(* Logix 5000 project; controller SX_V040001_C001 vendor 1 type 14 code 77 rev 16.22; software revision 16.04; part 15 of 35 *)
(* tags used below, declared in another part *)
   G_DInput : DINT[3];
   G_DOutput : DINT[3];
   louvre : INT[11];
   PARAMETER : INT[501];
(* MainProgram, continued *)

ROUTINE Louvre3Position   (* ladder *)
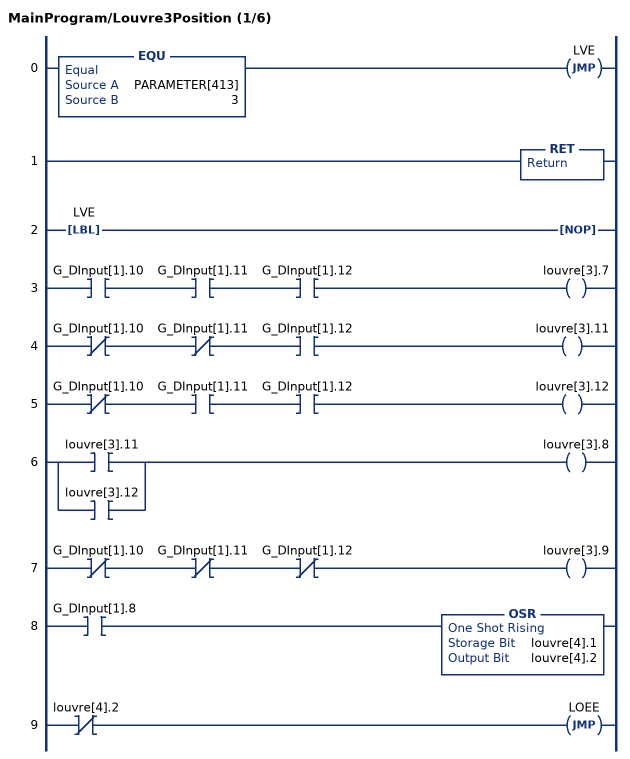
   0: EQU(PARAMETER[413],3)JMP(LVE);
   1: RET();
   2: LBL(LVE)NOP();
   3: XIC(G_DInput[1].10)XIC(G_DInput[1].11)XIC(G_DInput[1].12)OTE(louvre[3].7);
   4: XIO(G_DInput[1].10)XIO(G_DInput[1].11)XIC(G_DInput[1].12)OTE(louvre[3].11);
   5: XIO(G_DInput[1].10)XIC(G_DInput[1].11)XIC(G_DInput[1].12)OTE(louvre[3].12);
   6: [XIC(louvre[3].11) ,XIC(louvre[3].12) ]OTE(louvre[3].8);
   7: XIO(G_DInput[1].10)XIO(G_DInput[1].11)XIO(G_DInput[1].12)OTE(louvre[3].9);
   8: XIC(G_DInput[1].8)OSR(louvre[4].1,louvre[4].2);
   9: XIO(louvre[4].2)JMP(LOEE);
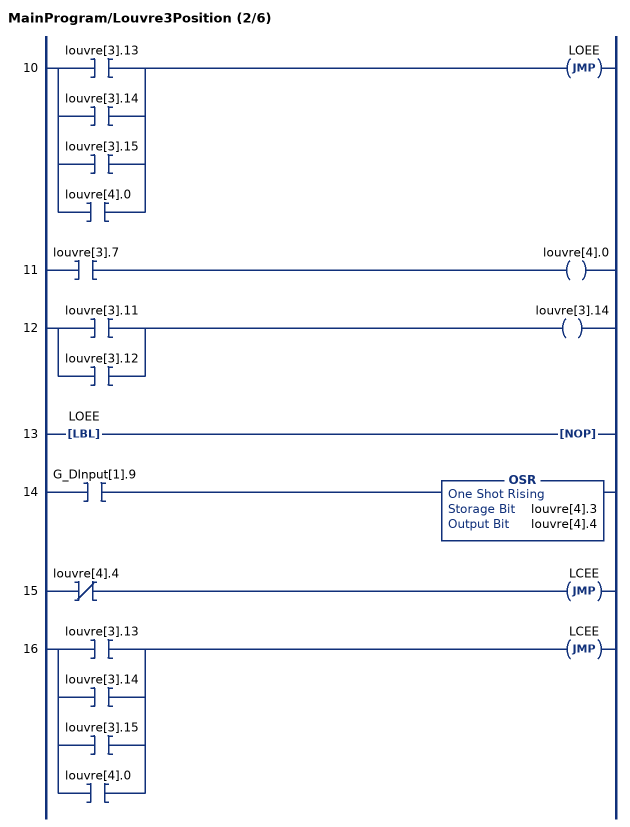
   10: [XIC(louvre[3].13) ,XIC(louvre[3].14) ,XIC(louvre[3].15) ,XIC(louvre[4].0) ]JMP(LOEE);
   11: XIC(louvre[3].7)OTE(louvre[4].0);
   12: [XIC(louvre[3].11) ,XIC(louvre[3].12) ]OTE(louvre[3].14);
   13: LBL(LOEE)NOP();
   14: XIC(G_DInput[1].9)OSR(louvre[4].3,louvre[4].4);
   15: XIO(louvre[4].4)JMP(LCEE);
   16: [XIC(louvre[3].13) ,XIC(louvre[3].14) ,XIC(louvre[3].15) ,XIC(louvre[4].0) ]JMP(LCEE);
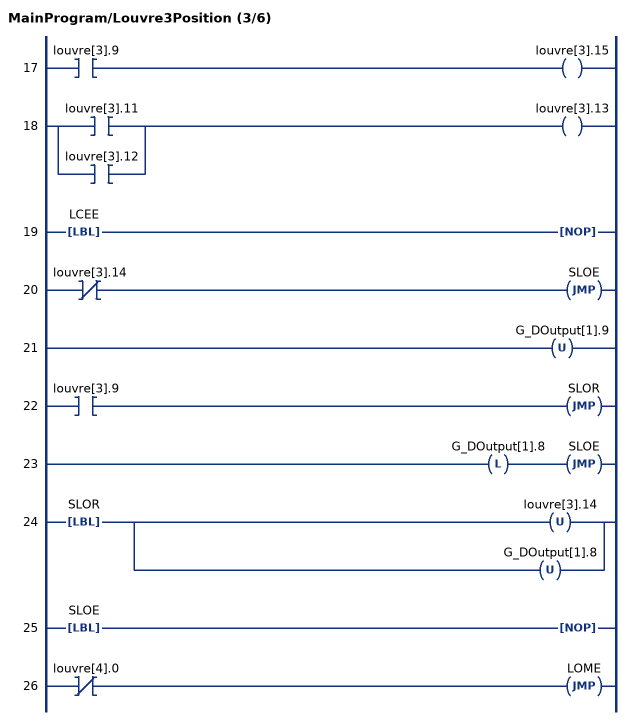
   17: XIC(louvre[3].9)OTE(louvre[3].15);
   18: [XIC(louvre[3].11) ,XIC(louvre[3].12) ]OTE(louvre[3].13);
   19: LBL(LCEE)NOP();
   20: XIO(louvre[3].14)JMP(SLOE);
   21: OTU(G_DOutput[1].9);
   22: XIC(louvre[3].9)JMP(SLOR);
   23: OTL(G_DOutput[1].8)JMP(SLOE);
   24: LBL(SLOR)[OTU(louvre[3].14) ,OTU(G_DOutput[1].8) ];
   25: LBL(SLOE)NOP();
   26: XIO(louvre[4].0)JMP(LOME);
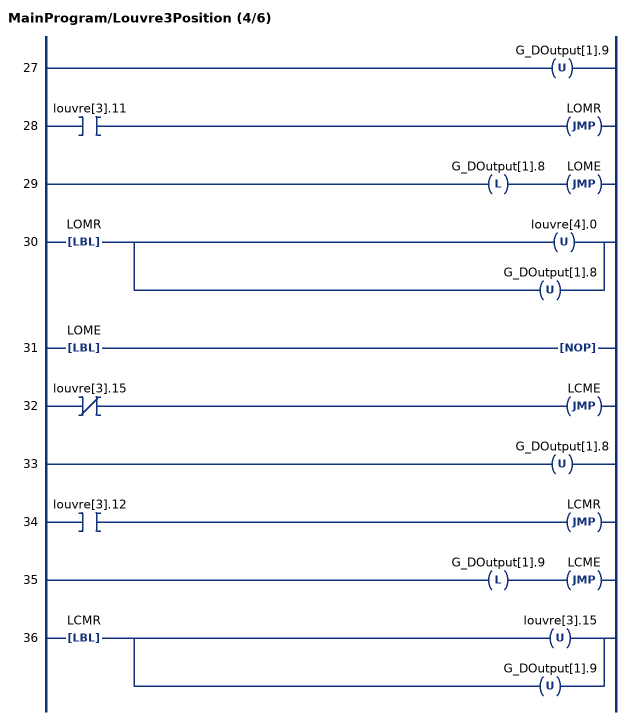
   27: OTU(G_DOutput[1].9);
   28: XIC(louvre[3].11)JMP(LOMR);
   29: OTL(G_DOutput[1].8)JMP(LOME);
   30: LBL(LOMR)[OTU(louvre[4].0) ,OTU(G_DOutput[1].8) ];
   31: LBL(LOME)NOP();
   32: XIO(louvre[3].15)JMP(LCME);
   33: OTU(G_DOutput[1].8);
   34: XIC(louvre[3].12)JMP(LCMR);
   35: OTL(G_DOutput[1].9)JMP(LCME);
   36: LBL(LCMR)[OTU(louvre[3].15) ,OTU(G_DOutput[1].9) ];
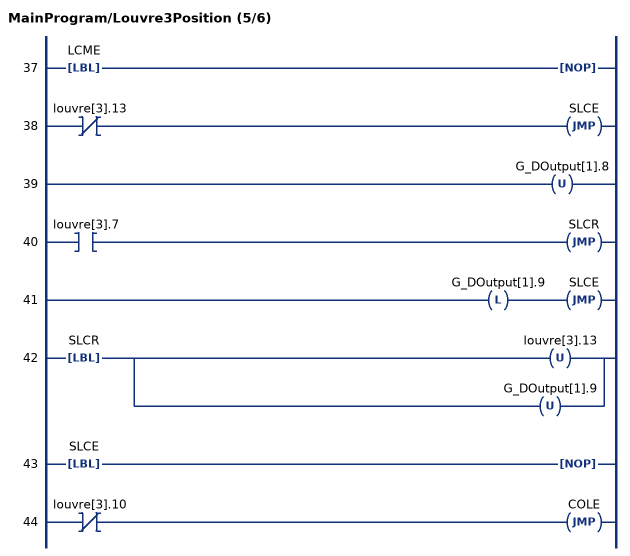
   37: LBL(LCME)NOP();
   38: XIO(louvre[3].13)JMP(SLCE);
   39: OTU(G_DOutput[1].8);
   40: XIC(louvre[3].7)JMP(SLCR);
   41: OTL(G_DOutput[1].9)JMP(SLCE);
   42: LBL(SLCR)[OTU(louvre[3].13) ,OTU(G_DOutput[1].9) ];
   43: LBL(SLCE)NOP();
   44: XIO(louvre[3].10)JMP(COLE);
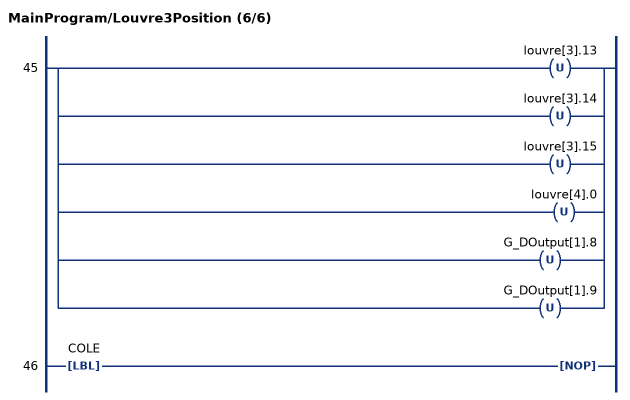
   45: [OTU(louvre[3].13) ,OTU(louvre[3].14) ,OTU(louvre[3].15) ,OTU(louvre[4].0) ,OTU(G_DOutput[1].8) ,OTU(G_DOutput[1].9) ];
   46: LBL(COLE)NOP();
END_ROUTINE

ROUTINE LouvreVariable   (* ladder *)
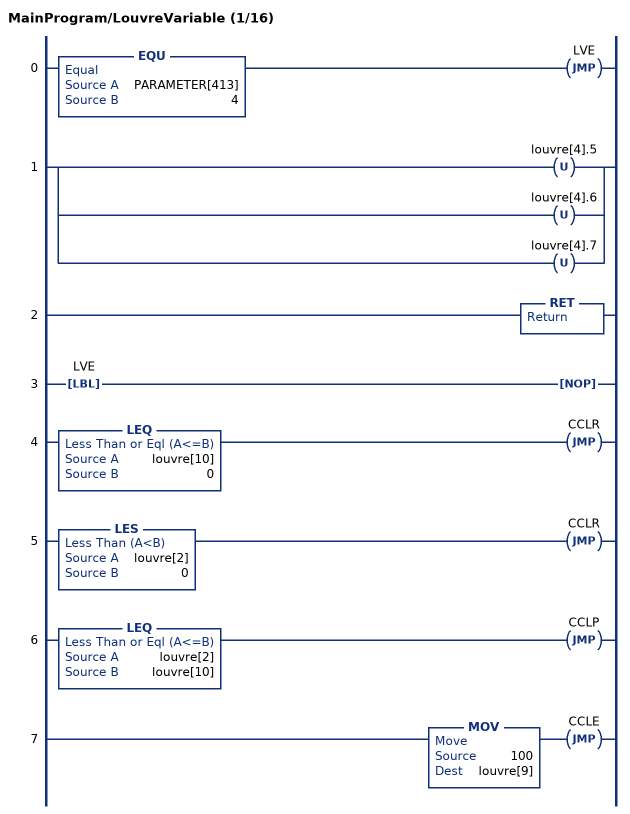
   0: EQU(PARAMETER[413],4)JMP(LVE);
   1: [OTU(louvre[4].5) ,OTU(louvre[4].6) ,OTU(louvre[4].7) ];
   2: RET();
   3: LBL(LVE)NOP();
   4: LEQ(louvre[10],0)JMP(CCLR);
   5: LES(louvre[2],0)JMP(CCLR);
   6: LEQ(louvre[2],louvre[10])JMP(CCLP);
   7: MOV(100,louvre[9])JMP(CCLE);
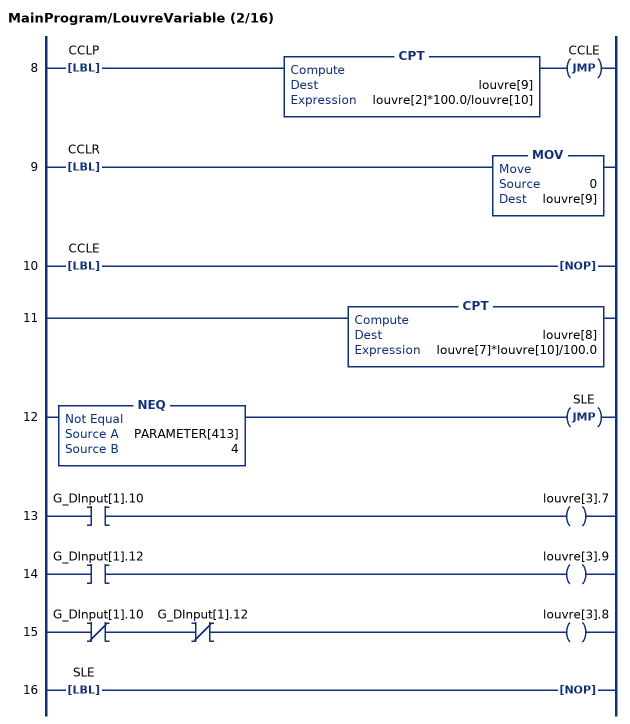
   8: LBL(CCLP)CPT(louvre[9],louvre[2]*100.0/louvre[10])JMP(CCLE);
   9: LBL(CCLR)MOV(0,louvre[9]);
   10: LBL(CCLE)NOP();
   11: CPT(louvre[8],louvre[7]*louvre[10]/100.0);
   12: NEQ(PARAMETER[413],4)JMP(SLE);
   13: XIC(G_DInput[1].10)OTE(louvre[3].7);
   14: XIC(G_DInput[1].12)OTE(louvre[3].9);
   15: XIO(G_DInput[1].10)XIO(G_DInput[1].12)OTE(louvre[3].8);
   16: LBL(SLE)NOP();
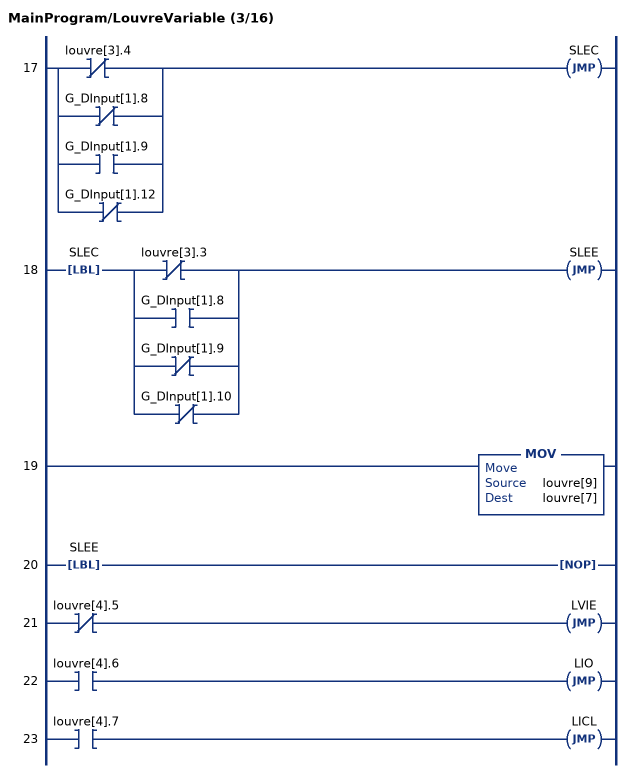
   17: [XIO(louvre[3].4) ,XIO(G_DInput[1].8) ,XIC(G_DInput[1].9) ,XIO(G_DInput[1].12) ]JMP(SLEC);
   18: LBL(SLEC)[XIO(louvre[3].3) ,XIC(G_DInput[1].8) ,XIO(G_DInput[1].9) ,XIO(G_DInput[1].10) ]JMP(SLEE);
   19: MOV(louvre[9],louvre[7]);
   20: LBL(SLEE)NOP();
   21: XIO(louvre[4].5)JMP(LVIE);
   22: XIC(louvre[4].6)JMP(LIO);
   23: XIC(louvre[4].7)JMP(LICL);
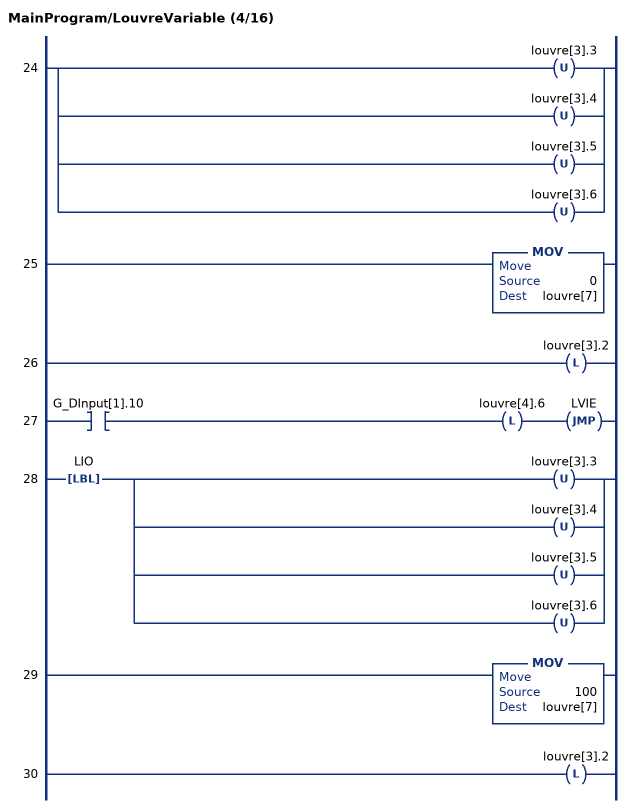
   24: [OTU(louvre[3].3) ,OTU(louvre[3].4) ,OTU(louvre[3].5) ,OTU(louvre[3].6) ];
   25: MOV(0,louvre[7]);
   26: OTL(louvre[3].2);
   27: XIC(G_DInput[1].10)OTL(louvre[4].6)JMP(LVIE);
   28: LBL(LIO)[OTU(louvre[3].3) ,OTU(louvre[3].4) ,OTU(louvre[3].5) ,OTU(louvre[3].6) ];
   29: MOV(100,louvre[7]);
   30: OTL(louvre[3].2);
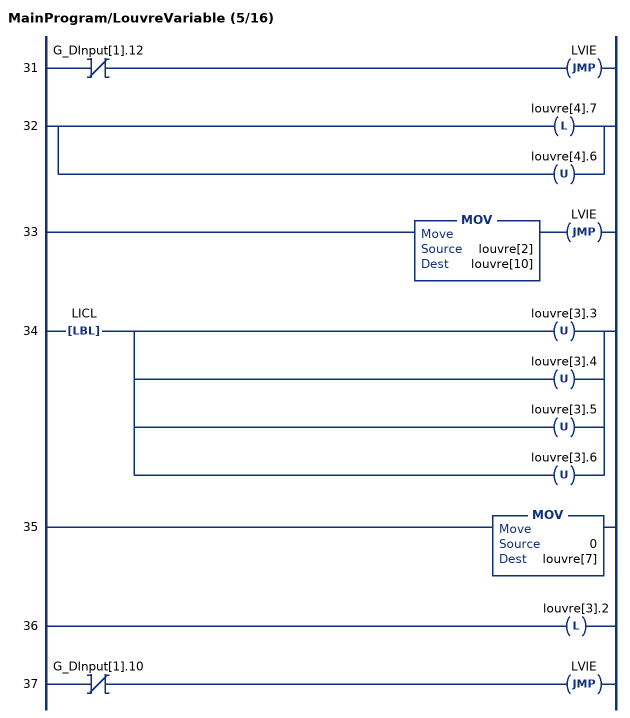
   31: XIO(G_DInput[1].12)JMP(LVIE);
   32: [OTL(louvre[4].7) ,OTU(louvre[4].6) ];
   33: MOV(louvre[2],louvre[10])JMP(LVIE);
   34: LBL(LICL)[OTU(louvre[3].3) ,OTU(louvre[3].4) ,OTU(louvre[3].5) ,OTU(louvre[3].6) ];
   35: MOV(0,louvre[7]);
   36: OTL(louvre[3].2);
   37: XIO(G_DInput[1].10)JMP(LVIE);
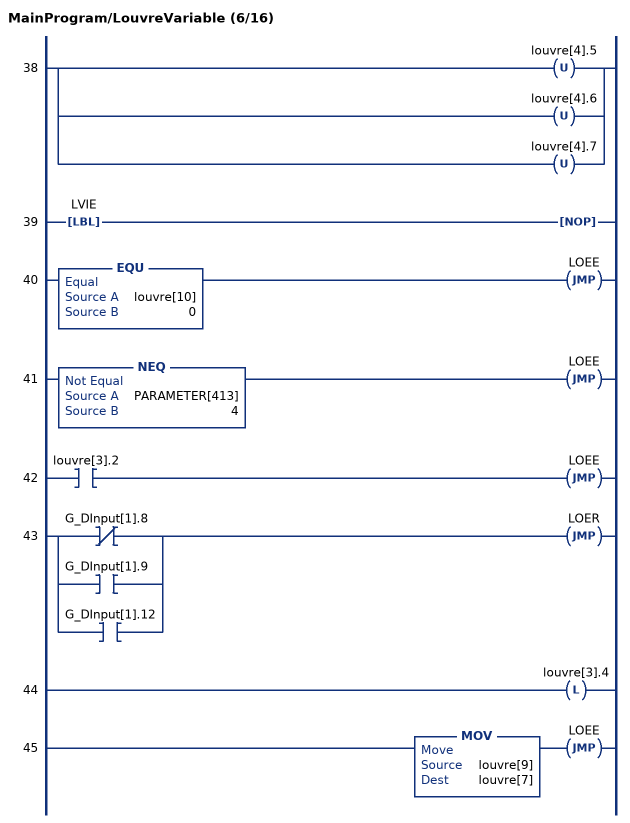
   38: [OTU(louvre[4].5) ,OTU(louvre[4].6) ,OTU(louvre[4].7) ];
   39: LBL(LVIE)NOP();
   40: EQU(louvre[10],0)JMP(LOEE);
   41: NEQ(PARAMETER[413],4)JMP(LOEE);
   42: XIC(louvre[3].2)JMP(LOEE);
   43: [XIO(G_DInput[1].8) ,XIC(G_DInput[1].9) ,XIC(G_DInput[1].12) ]JMP(LOER);
   44: OTL(louvre[3].4);
   45: MOV(louvre[9],louvre[7])JMP(LOEE);
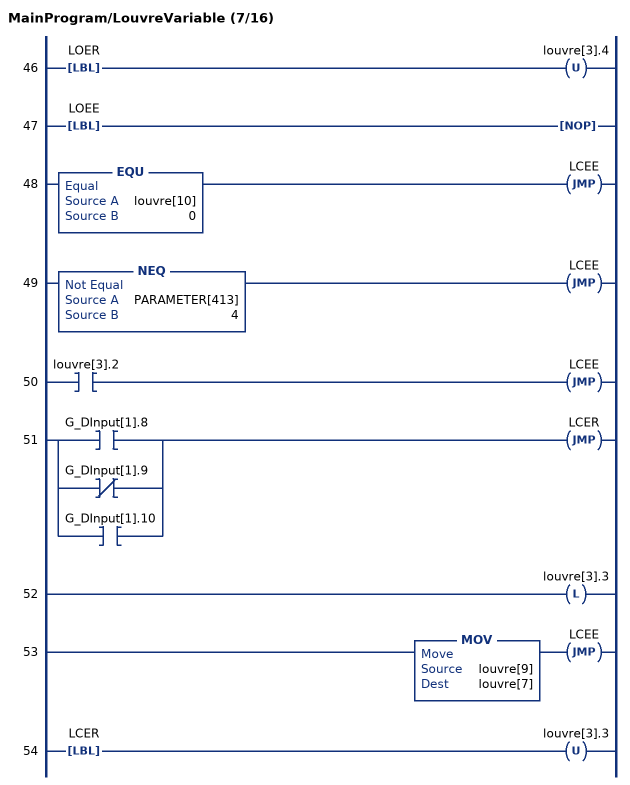
   46: LBL(LOER)OTU(louvre[3].4);
   47: LBL(LOEE)NOP();
   48: EQU(louvre[10],0)JMP(LCEE);
   49: NEQ(PARAMETER[413],4)JMP(LCEE);
   50: XIC(louvre[3].2)JMP(LCEE);
   51: [XIC(G_DInput[1].8) ,XIO(G_DInput[1].9) ,XIC(G_DInput[1].10) ]JMP(LCER);
   52: OTL(louvre[3].3);
   53: MOV(louvre[9],louvre[7])JMP(LCEE);
   54: LBL(LCER)OTU(louvre[3].3);
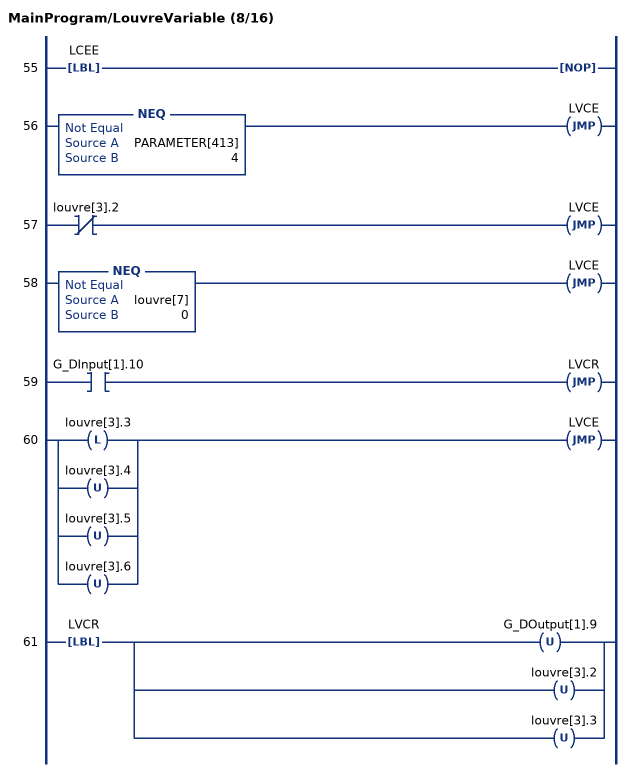
   55: LBL(LCEE)NOP();
   56: NEQ(PARAMETER[413],4)JMP(LVCE);
   57: XIO(louvre[3].2)JMP(LVCE);
   58: NEQ(louvre[7],0)JMP(LVCE);
   59: XIC(G_DInput[1].10)JMP(LVCR);
   60: [OTL(louvre[3].3) ,OTU(louvre[3].4) ,OTU(louvre[3].5) ,OTU(louvre[3].6) ]JMP(LVCE);
   61: LBL(LVCR)[OTU(G_DOutput[1].9) ,OTU(louvre[3].2) ,OTU(louvre[3].3) ];
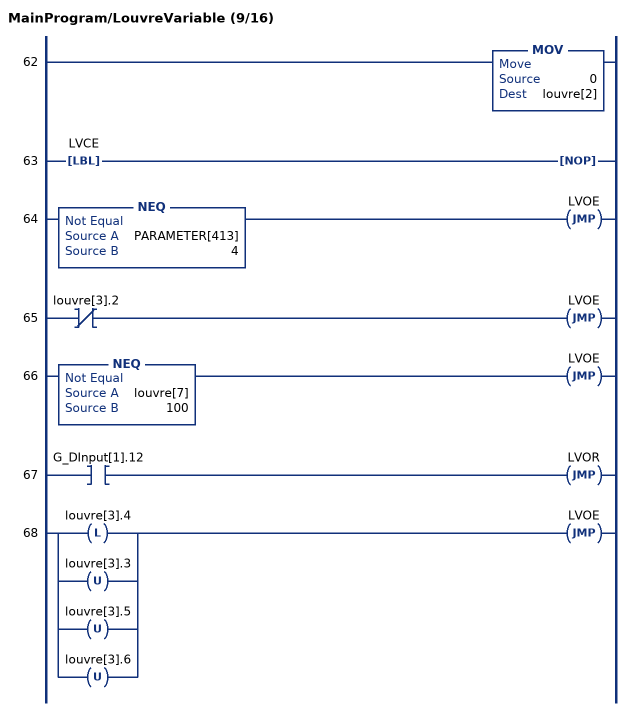
   62: MOV(0,louvre[2]);
   63: LBL(LVCE)NOP();
   64: NEQ(PARAMETER[413],4)JMP(LVOE);
   65: XIO(louvre[3].2)JMP(LVOE);
   66: NEQ(louvre[7],100)JMP(LVOE);
   67: XIC(G_DInput[1].12)JMP(LVOR);
   68: [OTL(louvre[3].4) ,OTU(louvre[3].3) ,OTU(louvre[3].5) ,OTU(louvre[3].6) ]JMP(LVOE);
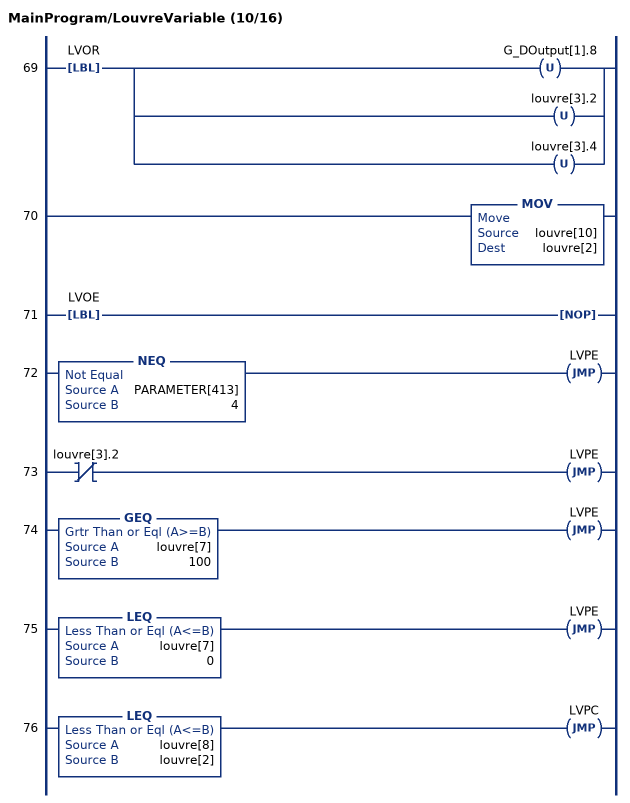
   69: LBL(LVOR)[OTU(G_DOutput[1].8) ,OTU(louvre[3].2) ,OTU(louvre[3].4) ];
   70: MOV(louvre[10],louvre[2]);
   71: LBL(LVOE)NOP();
   72: NEQ(PARAMETER[413],4)JMP(LVPE);
   73: XIO(louvre[3].2)JMP(LVPE);
   74: GEQ(louvre[7],100)JMP(LVPE);
   75: LEQ(louvre[7],0)JMP(LVPE);
   76: LEQ(louvre[8],louvre[2])JMP(LVPC);
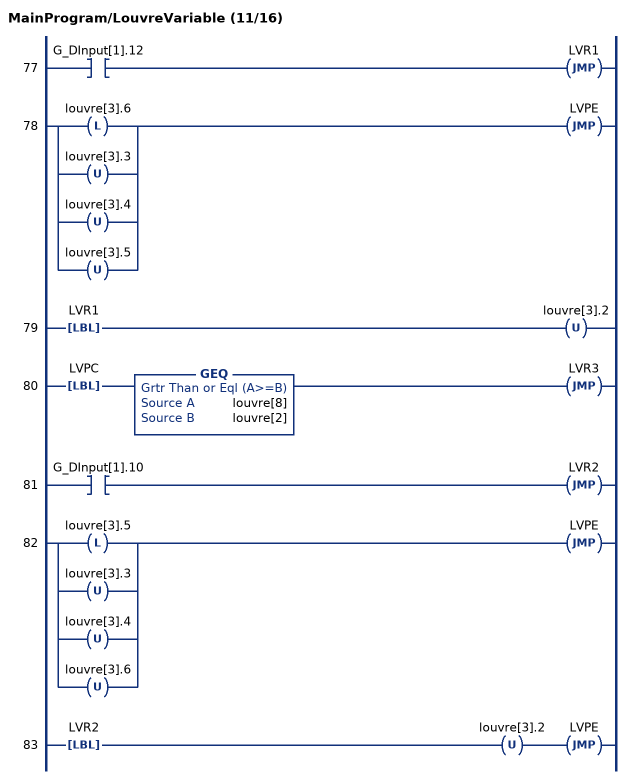
   77: XIC(G_DInput[1].12)JMP(LVR1);
   78: [OTL(louvre[3].6) ,OTU(louvre[3].3) ,OTU(louvre[3].4) ,OTU(louvre[3].5) ]JMP(LVPE);
   79: LBL(LVR1)OTU(louvre[3].2);
   80: LBL(LVPC)GEQ(louvre[8],louvre[2])JMP(LVR3);
   81: XIC(G_DInput[1].10)JMP(LVR2);
   82: [OTL(louvre[3].5) ,OTU(louvre[3].3) ,OTU(louvre[3].4) ,OTU(louvre[3].6) ]JMP(LVPE);
   83: LBL(LVR2)OTU(louvre[3].2)JMP(LVPE);
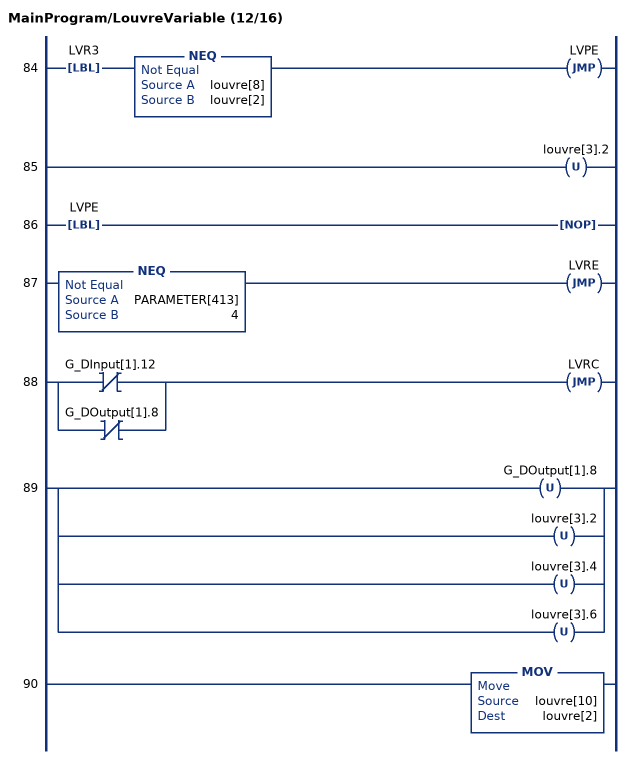
   84: LBL(LVR3)NEQ(louvre[8],louvre[2])JMP(LVPE);
   85: OTU(louvre[3].2);
   86: LBL(LVPE)NOP();
   87: NEQ(PARAMETER[413],4)JMP(LVRE);
   88: [XIO(G_DInput[1].12) ,XIO(G_DOutput[1].8) ]JMP(LVRC);
   89: [OTU(G_DOutput[1].8) ,OTU(louvre[3].2) ,OTU(louvre[3].4) ,OTU(louvre[3].6) ];
   90: MOV(louvre[10],louvre[2]);
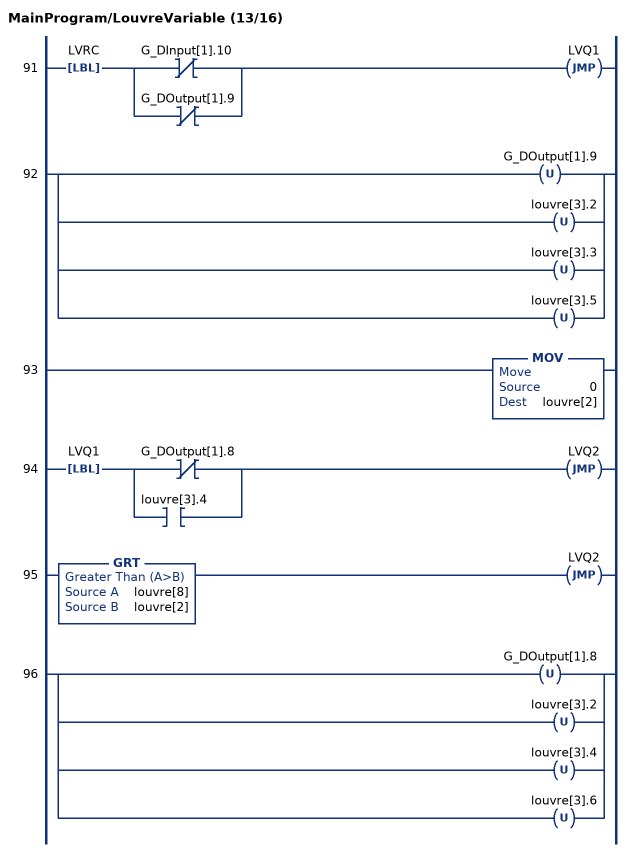
   91: LBL(LVRC)[XIO(G_DInput[1].10) ,XIO(G_DOutput[1].9) ]JMP(LVQ1);
   92: [OTU(G_DOutput[1].9) ,OTU(louvre[3].2) ,OTU(louvre[3].3) ,OTU(louvre[3].5) ];
   93: MOV(0,louvre[2]);
   94: LBL(LVQ1)[XIO(G_DOutput[1].8) ,XIC(louvre[3].4) ]JMP(LVQ2);
   95: GRT(louvre[8],louvre[2])JMP(LVQ2);
   96: [OTU(G_DOutput[1].8) ,OTU(louvre[3].2) ,OTU(louvre[3].4) ,OTU(louvre[3].6) ];
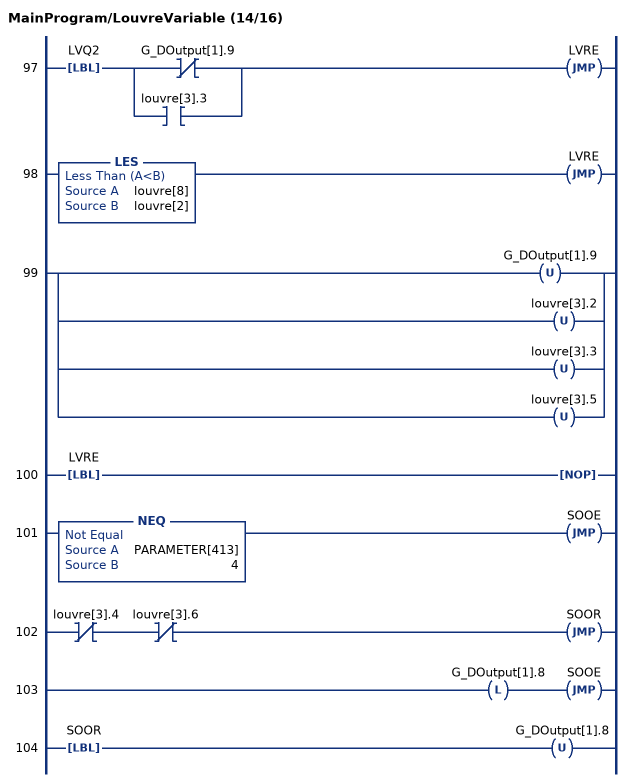
   97: LBL(LVQ2)[XIO(G_DOutput[1].9) ,XIC(louvre[3].3) ]JMP(LVRE);
   98: LES(louvre[8],louvre[2])JMP(LVRE);
   99: [OTU(G_DOutput[1].9) ,OTU(louvre[3].2) ,OTU(louvre[3].3) ,OTU(louvre[3].5) ];
   100: LBL(LVRE)NOP();
   101: NEQ(PARAMETER[413],4)JMP(SOOE);
   102: XIO(louvre[3].4)XIO(louvre[3].6)JMP(SOOR);
   103: OTL(G_DOutput[1].8)JMP(SOOE);
   104: LBL(SOOR)OTU(G_DOutput[1].8);
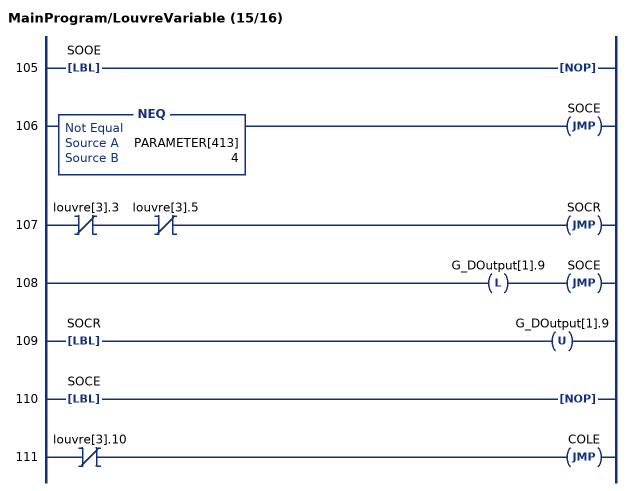
   105: LBL(SOOE)NOP();
   106: NEQ(PARAMETER[413],4)JMP(SOCE);
   107: XIO(louvre[3].3)XIO(louvre[3].5)JMP(SOCR);
   108: OTL(G_DOutput[1].9)JMP(SOCE);
   109: LBL(SOCR)OTU(G_DOutput[1].9);
   110: LBL(SOCE)NOP();
   111: XIO(louvre[3].10)JMP(COLE);
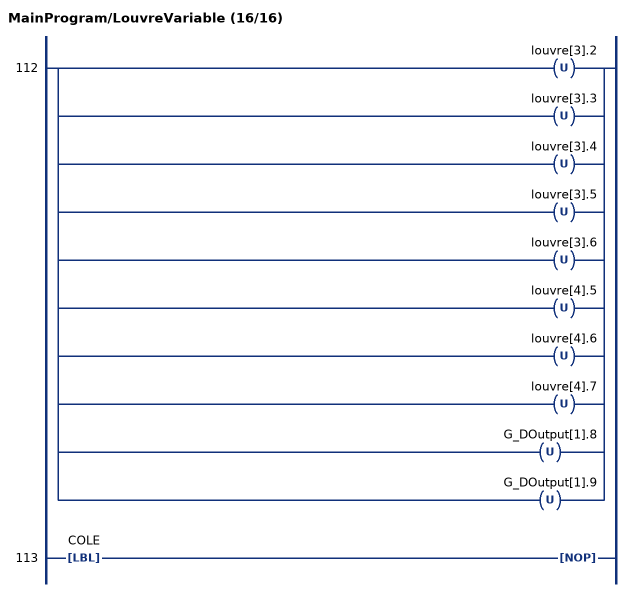
   112: [OTU(louvre[3].2) ,OTU(louvre[3].3) ,OTU(louvre[3].4) ,OTU(louvre[3].5) ,OTU(louvre[3].6) ,OTU(louvre[4].5) ,OTU(louvre[4].6) ,OTU(louvre[4].7) ,OTU(G_DOutput[1].8) ,OTU(G_DOutput[1].9) ];
   113: LBL(COLE)NOP();
END_ROUTINE
